(*
version 1.5	2. jan. 2012
programmer 	hugo
tested by	oscat

this function will insert a string at a given position in a buffer.
the function needs to be called:	_buffer_init(adr("array"),sizeof("array"),init);
this function will manipulate a given array.
the function manipulates the original array, it returnes the next position after the input string when finished.
because this function works with pointers its very time efficient and it needs no extra memory.

*)
FUNCTION _BUFFER_INSERT : INT
VAR_INPUT
	STR : STRING(STRING_LENGTH);
	POS : INT;
	PT : POINTER TO ARRAY[0..32767] OF BYTE;
	SIZE : UINT;
END_VAR
VAR
	end : INT;
	lx: INT;
	i: INT;
END_VAR

lx := LEN(str);
end := pos + lx;
(* first move the upper part of the buffer to make space for the string *)
FOR i := UINT_TO_INT(size) - 1 TO end BY -1 DO
	pt^[i] := pt^[i-lx];
END_FOR;
(* copy the string *)
_BUFFER_INSERT := _STRING_TO_BUFFER(str, pos, PT, size);


(* revision History
hm 	9. mar. 2008	rev 1.0
	original version

hm	16. mar. 2008	rev 1.1
	changed type of input size to uint

hm	13. may. 2008	rev 1.2
	changed type of pointer to array[1..32767]
	changed size of string to STRING_LENGTH

hm	23. mar. 2009	rev 1.3
	avoid writing to input pos

hm	12. nov. 2009	rev 1.4
	code optimized

hm 2. jan 2012	rev 1.5
	function now returns the next position after the input string

*)

END_FUNCTION

(* stored: Version 1.1.0.1
   POU _BUFFER_INSERT: Id {125d3592-a908-4550-b6ec-b75c1e0fe3fd}, SpecialFunc None *)
